
FUNCTION CB_dword_to_dint : DINT

TITLE = ' Convert a double word into a Double integer '
VERSION : '1.0'
AUTHOR  : CB
NAME    : DworToDi
FAMILY  : TNI

VAR_INPUT
    IN : DWORD;
END_VAR

VAR_TEMP

END_VAR

BEGIN

CB_dword_to_dint := DWORD_TO_DINT(IN);

END_FUNCTION
